FUNCTION_BLOCK FB_Test
VAR_INPUT
END_VAR
VAR_OUTPUT
END_VAR
VAR
END_VAR

END_FUNCTION_BLOCK

(* stored: Version 1.1.0.1, ProductVersion 3.1.4024.5
   POU FB_Test: Id {b756cabd-24af-4ae0-a617-3a5bcf37e93a}, SpecialFunc None *)
